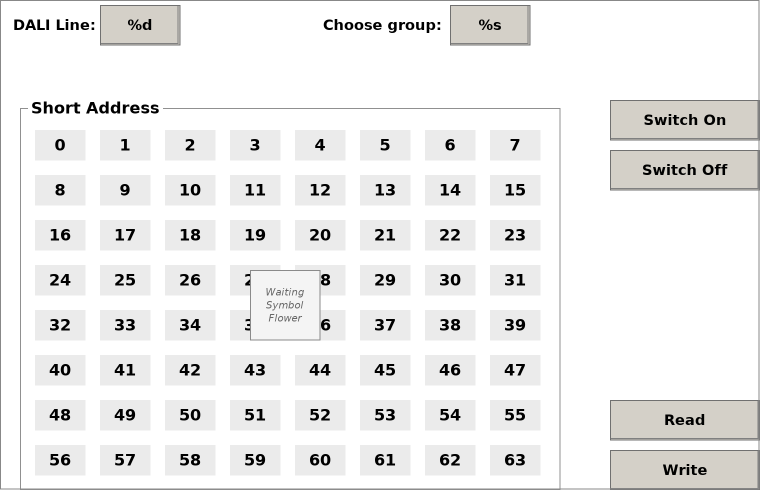
VISUALIZATION Visu_Part102Groups  // 760x490
    GroupBox (20,100 540x390), "Short Address"
        Textfield (15,30 50x30), "0", colour toggle: DALI_Commissioning.fbPart102Groups.aShowAlarmState[0] = TRUE, invisible if: DALI_Commissioning.fbPart102Groups.aActivateButton[0] = FALSE, input disabled if: DALI_Commissioning.fbPart102Groups.aActivateButton[0] = FALSE
            OnMouseClick: execute { DALI_Commissioning.fbPart102Groups.aButtonClick[0] := TRUE; }
        Textfield (80,30 50x30), "1", colour toggle: DALI_Commissioning.fbPart102Groups.aShowAlarmState[1] = TRUE, invisible if: DALI_Commissioning.fbPart102Groups.aActivateButton[1] = FALSE, input disabled if: DALI_Commissioning.fbPart102Groups.aActivateButton[1] = FALSE
            OnMouseClick: execute { DALI_Commissioning.fbPart102Groups.aButtonClick[1] := TRUE; }
        Textfield (145,30 50x30), "2", colour toggle: DALI_Commissioning.fbPart102Groups.aShowAlarmState[2] = TRUE, invisible if: DALI_Commissioning.fbPart102Groups.aActivateButton[2] = FALSE, input disabled if: DALI_Commissioning.fbPart102Groups.aActivateButton[2] = FALSE
            OnMouseClick: execute { DALI_Commissioning.fbPart102Groups.aButtonClick[2] := TRUE; }
        Textfield (210,30 50x30), "3", colour toggle: DALI_Commissioning.fbPart102Groups.aShowAlarmState[3] = TRUE, invisible if: DALI_Commissioning.fbPart102Groups.aActivateButton[3] = FALSE, input disabled if: DALI_Commissioning.fbPart102Groups.aActivateButton[3] = FALSE
            OnMouseClick: execute { DALI_Commissioning.fbPart102Groups.aButtonClick[3] := TRUE; }
        Textfield (275,30 50x30), "4", colour toggle: DALI_Commissioning.fbPart102Groups.aShowAlarmState[4] = TRUE, invisible if: DALI_Commissioning.fbPart102Groups.aActivateButton[4] = FALSE, input disabled if: DALI_Commissioning.fbPart102Groups.aActivateButton[4] = FALSE
            OnMouseClick: execute { DALI_Commissioning.fbPart102Groups.aButtonClick[4] := TRUE; }
        Textfield (340,30 50x30), "5", colour toggle: DALI_Commissioning.fbPart102Groups.aShowAlarmState[5] = TRUE, invisible if: DALI_Commissioning.fbPart102Groups.aActivateButton[5] = FALSE, input disabled if: DALI_Commissioning.fbPart102Groups.aActivateButton[5] = FALSE
            OnMouseClick: execute { DALI_Commissioning.fbPart102Groups.aButtonClick[5] := TRUE; }
        Textfield (405,30 50x30), "6", colour toggle: DALI_Commissioning.fbPart102Groups.aShowAlarmState[6] = TRUE, invisible if: DALI_Commissioning.fbPart102Groups.aActivateButton[6] = FALSE, input disabled if: DALI_Commissioning.fbPart102Groups.aActivateButton[6] = FALSE
            OnMouseClick: execute { DALI_Commissioning.fbPart102Groups.aButtonClick[6] := TRUE; }
        Textfield (470,30 50x30), "7", colour toggle: DALI_Commissioning.fbPart102Groups.aShowAlarmState[7] = TRUE, invisible if: DALI_Commissioning.fbPart102Groups.aActivateButton[7] = FALSE, input disabled if: DALI_Commissioning.fbPart102Groups.aActivateButton[7] = FALSE
            OnMouseClick: execute { DALI_Commissioning.fbPart102Groups.aButtonClick[7] := TRUE; }
        Textfield (15,75 50x30), "8", colour toggle: DALI_Commissioning.fbPart102Groups.aShowAlarmState[8] = TRUE, invisible if: DALI_Commissioning.fbPart102Groups.aActivateButton[8] = FALSE, input disabled if: DALI_Commissioning.fbPart102Groups.aActivateButton[8] = FALSE
            OnMouseClick: execute { DALI_Commissioning.fbPart102Groups.aButtonClick[8] := TRUE; }
        Textfield (80,75 50x30), "9", colour toggle: DALI_Commissioning.fbPart102Groups.aShowAlarmState[9] = TRUE, invisible if: DALI_Commissioning.fbPart102Groups.aActivateButton[9] = FALSE, input disabled if: DALI_Commissioning.fbPart102Groups.aActivateButton[9] = FALSE
            OnMouseClick: execute { DALI_Commissioning.fbPart102Groups.aButtonClick[9] := TRUE; }
        Textfield (145,75 50x30), "10", colour toggle: DALI_Commissioning.fbPart102Groups.aShowAlarmState[10] = TRUE, invisible if: DALI_Commissioning.fbPart102Groups.aActivateButton[10] = FALSE, input disabled if: DALI_Commissioning.fbPart102Groups.aActivateButton[10] = FALSE
            OnMouseClick: execute { DALI_Commissioning.fbPart102Groups.aButtonClick[10] := TRUE; }
        Textfield (210,75 50x30), "11", colour toggle: DALI_Commissioning.fbPart102Groups.aShowAlarmState[11] = TRUE, invisible if: DALI_Commissioning.fbPart102Groups.aActivateButton[11] = FALSE, input disabled if: DALI_Commissioning.fbPart102Groups.aActivateButton[11] = FALSE
            OnMouseClick: execute { DALI_Commissioning.fbPart102Groups.aButtonClick[11] := TRUE; }
        Textfield (275,75 50x30), "12", colour toggle: DALI_Commissioning.fbPart102Groups.aShowAlarmState[12] = TRUE, invisible if: DALI_Commissioning.fbPart102Groups.aActivateButton[12] = FALSE, input disabled if: DALI_Commissioning.fbPart102Groups.aActivateButton[12] = FALSE
            OnMouseClick: execute { DALI_Commissioning.fbPart102Groups.aButtonClick[12] := TRUE; }
        Textfield (340,75 50x30), "13", colour toggle: DALI_Commissioning.fbPart102Groups.aShowAlarmState[13] = TRUE, invisible if: DALI_Commissioning.fbPart102Groups.aActivateButton[13] = FALSE, input disabled if: DALI_Commissioning.fbPart102Groups.aActivateButton[13] = FALSE
            OnMouseClick: execute { DALI_Commissioning.fbPart102Groups.aButtonClick[13] := TRUE; }
        Textfield (405,75 50x30), "14", colour toggle: DALI_Commissioning.fbPart102Groups.aShowAlarmState[14] = TRUE, invisible if: DALI_Commissioning.fbPart102Groups.aActivateButton[14] = FALSE, input disabled if: DALI_Commissioning.fbPart102Groups.aActivateButton[14] = FALSE
            OnMouseClick: execute { DALI_Commissioning.fbPart102Groups.aButtonClick[14] := TRUE; }
        Textfield (470,75 50x30), "15", colour toggle: DALI_Commissioning.fbPart102Groups.aShowAlarmState[15] = TRUE, invisible if: DALI_Commissioning.fbPart102Groups.aActivateButton[15] = FALSE, input disabled if: DALI_Commissioning.fbPart102Groups.aActivateButton[15] = FALSE
            OnMouseClick: execute { DALI_Commissioning.fbPart102Groups.aButtonClick[15] := TRUE; }
        Textfield (15,120 50x30), "16", colour toggle: DALI_Commissioning.fbPart102Groups.aShowAlarmState[16] = TRUE, invisible if: DALI_Commissioning.fbPart102Groups.aActivateButton[16] = FALSE, input disabled if: DALI_Commissioning.fbPart102Groups.aActivateButton[16] = FALSE
            OnMouseClick: execute { DALI_Commissioning.fbPart102Groups.aButtonClick[16] := TRUE; }
        Textfield (80,120 50x30), "17", colour toggle: DALI_Commissioning.fbPart102Groups.aShowAlarmState[17] = TRUE, invisible if: DALI_Commissioning.fbPart102Groups.aActivateButton[17] = FALSE, input disabled if: DALI_Commissioning.fbPart102Groups.aActivateButton[17] = FALSE
            OnMouseClick: execute { DALI_Commissioning.fbPart102Groups.aButtonClick[17] := TRUE; }
        Textfield (145,120 50x30), "18", colour toggle: DALI_Commissioning.fbPart102Groups.aShowAlarmState[18] = TRUE, invisible if: DALI_Commissioning.fbPart102Groups.aActivateButton[18] = FALSE, input disabled if: DALI_Commissioning.fbPart102Groups.aActivateButton[18] = FALSE
            OnMouseClick: execute { DALI_Commissioning.fbPart102Groups.aButtonClick[18] := TRUE; }
        Textfield (210,120 50x30), "19", colour toggle: DALI_Commissioning.fbPart102Groups.aShowAlarmState[19] = TRUE, invisible if: DALI_Commissioning.fbPart102Groups.aActivateButton[19] = FALSE, input disabled if: DALI_Commissioning.fbPart102Groups.aActivateButton[19] = FALSE
            OnMouseClick: execute { DALI_Commissioning.fbPart102Groups.aButtonClick[19] := TRUE; }
        Textfield (275,120 50x30), "20", colour toggle: DALI_Commissioning.fbPart102Groups.aShowAlarmState[20] = TRUE, invisible if: DALI_Commissioning.fbPart102Groups.aActivateButton[20] = FALSE, input disabled if: DALI_Commissioning.fbPart102Groups.aActivateButton[20] = FALSE
            OnMouseClick: execute { DALI_Commissioning.fbPart102Groups.aButtonClick[20] := TRUE; }
        Textfield (340,120 50x30), "21", colour toggle: DALI_Commissioning.fbPart102Groups.aShowAlarmState[21] = TRUE, invisible if: DALI_Commissioning.fbPart102Groups.aActivateButton[21] = FALSE, input disabled if: DALI_Commissioning.fbPart102Groups.aActivateButton[21] = FALSE
            OnMouseClick: execute { DALI_Commissioning.fbPart102Groups.aButtonClick[21] := TRUE; }
        Textfield (405,120 50x30), "22", colour toggle: DALI_Commissioning.fbPart102Groups.aShowAlarmState[22] = TRUE, invisible if: DALI_Commissioning.fbPart102Groups.aActivateButton[22] = FALSE, input disabled if: DALI_Commissioning.fbPart102Groups.aActivateButton[22] = FALSE
            OnMouseClick: execute { DALI_Commissioning.fbPart102Groups.aButtonClick[22] := TRUE; }
        Textfield (470,120 50x30), "23", colour toggle: DALI_Commissioning.fbPart102Groups.aShowAlarmState[23] = TRUE, invisible if: DALI_Commissioning.fbPart102Groups.aActivateButton[23] = FALSE, input disabled if: DALI_Commissioning.fbPart102Groups.aActivateButton[23] = FALSE
            OnMouseClick: execute { DALI_Commissioning.fbPart102Groups.aButtonClick[23] := TRUE; }
        Textfield (15,165 50x30), "24", colour toggle: DALI_Commissioning.fbPart102Groups.aShowAlarmState[24] = TRUE, invisible if: DALI_Commissioning.fbPart102Groups.aDeviceGroupState[24] = 0, input disabled if: DALI_Commissioning.fbPart102Groups.aDeviceGroupState[24] = 0
            OnMouseClick: execute { DALI_Commissioning.fbPart102Groups.aButtonClick[24] := TRUE; }
        Textfield (80,165 50x30), "25", colour toggle: DALI_Commissioning.fbPart102Groups.aShowAlarmState[25] = TRUE, invisible if: DALI_Commissioning.fbPart102Groups.aActivateButton[25] = FALSE, input disabled if: DALI_Commissioning.fbPart102Groups.aActivateButton[25] = FALSE
            OnMouseClick: execute { DALI_Commissioning.fbPart102Groups.aButtonClick[25] := TRUE; }
        Textfield (145,165 50x30), "26", colour toggle: DALI_Commissioning.fbPart102Groups.aShowAlarmState[26] = TRUE, invisible if: DALI_Commissioning.fbPart102Groups.aActivateButton[26] = FALSE, input disabled if: DALI_Commissioning.fbPart102Groups.aActivateButton[26] = FALSE
            OnMouseClick: execute { DALI_Commissioning.fbPart102Groups.aButtonClick[26] := TRUE; }
        Textfield (210,165 50x30), "27", colour toggle: DALI_Commissioning.fbPart102Groups.aShowAlarmState[27] = TRUE, invisible if: DALI_Commissioning.fbPart102Groups.aActivateButton[27] = FALSE, input disabled if: DALI_Commissioning.fbPart102Groups.aActivateButton[27] = FALSE
            OnMouseClick: execute { DALI_Commissioning.fbPart102Groups.aButtonClick[27] := TRUE; }
        Textfield (275,165 50x30), "28", colour toggle: DALI_Commissioning.fbPart102Groups.aShowAlarmState[28] = TRUE, invisible if: DALI_Commissioning.fbPart102Groups.aActivateButton[28] = FALSE, input disabled if: DALI_Commissioning.fbPart102Groups.aActivateButton[28] = FALSE
            OnMouseClick: execute { DALI_Commissioning.fbPart102Groups.aButtonClick[28] := TRUE; }
        Textfield (340,165 50x30), "29", colour toggle: DALI_Commissioning.fbPart102Groups.aShowAlarmState[29] = TRUE, invisible if: DALI_Commissioning.fbPart102Groups.aActivateButton[29] = FALSE, input disabled if: DALI_Commissioning.fbPart102Groups.aActivateButton[29] = FALSE
            OnMouseClick: execute { DALI_Commissioning.fbPart102Groups.aButtonClick[29] := TRUE; }
        Textfield (405,165 50x30), "30", colour toggle: DALI_Commissioning.fbPart102Groups.aShowAlarmState[30] = TRUE, invisible if: DALI_Commissioning.fbPart102Groups.aActivateButton[30] = FALSE, input disabled if: DALI_Commissioning.fbPart102Groups.aActivateButton[30] = FALSE
            OnMouseClick: execute { DALI_Commissioning.fbPart102Groups.aButtonClick[30] := TRUE; }
        Textfield (470,165 50x30), "31", colour toggle: DALI_Commissioning.fbPart102Groups.aShowAlarmState[31] = TRUE, invisible if: DALI_Commissioning.fbPart102Groups.aActivateButton[31] = FALSE, input disabled if: DALI_Commissioning.fbPart102Groups.aActivateButton[31] = FALSE
            OnMouseClick: execute { DALI_Commissioning.fbPart102Groups.aButtonClick[31] := TRUE; }
        Textfield (15,210 50x30), "32", colour toggle: DALI_Commissioning.fbPart102Groups.aShowAlarmState[32] = TRUE, invisible if: DALI_Commissioning.fbPart102Groups.aActivateButton[32] = FALSE, input disabled if: DALI_Commissioning.fbPart102Groups.aActivateButton[32] = FALSE
            OnMouseClick: execute { DALI_Commissioning.fbPart102Groups.aButtonClick[32] := TRUE; }
        Textfield (80,210 50x30), "33", colour toggle: DALI_Commissioning.fbPart102Groups.aShowAlarmState[33] = TRUE, invisible if: DALI_Commissioning.fbPart102Groups.aActivateButton[33] = FALSE, input disabled if: DALI_Commissioning.fbPart102Groups.aActivateButton[33] = FALSE
            OnMouseClick: execute { DALI_Commissioning.fbPart102Groups.aButtonClick[33] := TRUE; }
        Textfield (145,210 50x30), "34", colour toggle: DALI_Commissioning.fbPart102Groups.aShowAlarmState[34] = TRUE, invisible if: DALI_Commissioning.fbPart102Groups.aActivateButton[34] = FALSE, input disabled if: DALI_Commissioning.fbPart102Groups.aActivateButton[34] = FALSE
            OnMouseClick: execute { DALI_Commissioning.fbPart102Groups.aButtonClick[34] := TRUE; }
        Textfield (210,210 50x30), "35", colour toggle: DALI_Commissioning.fbPart102Groups.aShowAlarmState[35] = TRUE, invisible if: DALI_Commissioning.fbPart102Groups.aActivateButton[35] = FALSE, input disabled if: DALI_Commissioning.fbPart102Groups.aActivateButton[35] = FALSE
            OnMouseClick: execute { DALI_Commissioning.fbPart102Groups.aButtonClick[35] := TRUE; }
        Textfield (275,210 50x30), "36", colour toggle: DALI_Commissioning.fbPart102Groups.aShowAlarmState[36] = TRUE, invisible if: DALI_Commissioning.fbPart102Groups.aActivateButton[36] = FALSE, input disabled if: DALI_Commissioning.fbPart102Groups.aActivateButton[36] = FALSE
            OnMouseClick: execute { DALI_Commissioning.fbPart102Groups.aButtonClick[36] := TRUE; }
        Textfield (340,210 50x30), "37", colour toggle: DALI_Commissioning.fbPart102Groups.aShowAlarmState[37] = TRUE, invisible if: DALI_Commissioning.fbPart102Groups.aActivateButton[37] = FALSE, input disabled if: DALI_Commissioning.fbPart102Groups.aActivateButton[37] = FALSE
            OnMouseClick: execute { DALI_Commissioning.fbPart102Groups.aButtonClick[37] := TRUE; }
        Textfield (405,210 50x30), "38", colour toggle: DALI_Commissioning.fbPart102Groups.aShowAlarmState[38] = TRUE, invisible if: DALI_Commissioning.fbPart102Groups.aActivateButton[38] = FALSE, input disabled if: DALI_Commissioning.fbPart102Groups.aActivateButton[38] = FALSE
            OnMouseClick: execute { DALI_Commissioning.fbPart102Groups.aButtonClick[38] := TRUE; }
        Textfield (470,210 50x30), "39", colour toggle: DALI_Commissioning.fbPart102Groups.aShowAlarmState[39] = TRUE, invisible if: DALI_Commissioning.fbPart102Groups.aActivateButton[39] = FALSE, input disabled if: DALI_Commissioning.fbPart102Groups.aActivateButton[39] = FALSE
            OnMouseClick: execute { DALI_Commissioning.fbPart102Groups.aButtonClick[39] := TRUE; }
        Textfield (15,255 50x30), "40", colour toggle: DALI_Commissioning.fbPart102Groups.aShowAlarmState[40] = TRUE, invisible if: DALI_Commissioning.fbPart102Groups.aActivateButton[40] = FALSE, input disabled if: DALI_Commissioning.fbPart102Groups.aActivateButton[40] = FALSE
            OnMouseClick: execute { DALI_Commissioning.fbPart102Groups.aButtonClick[40] := TRUE; }
        Textfield (80,255 50x30), "41", colour toggle: DALI_Commissioning.fbPart102Groups.aShowAlarmState[41] = TRUE, invisible if: DALI_Commissioning.fbPart102Groups.aActivateButton[41] = FALSE, input disabled if: DALI_Commissioning.fbPart102Groups.aActivateButton[41] = FALSE
            OnMouseClick: execute { DALI_Commissioning.fbPart102Groups.aButtonClick[41] := TRUE; }
        Textfield (145,255 50x30), "42", colour toggle: DALI_Commissioning.fbPart102Groups.aShowAlarmState[42] = TRUE, invisible if: DALI_Commissioning.fbPart102Groups.aActivateButton[42] = FALSE, input disabled if: DALI_Commissioning.fbPart102Groups.aActivateButton[42] = FALSE
            OnMouseClick: execute { DALI_Commissioning.fbPart102Groups.aButtonClick[42] := TRUE; }
        Textfield (210,255 50x30), "43", colour toggle: DALI_Commissioning.fbPart102Groups.aShowAlarmState[43] = TRUE, invisible if: DALI_Commissioning.fbPart102Groups.aActivateButton[43] = FALSE, input disabled if: DALI_Commissioning.fbPart102Groups.aActivateButton[43] = FALSE
            OnMouseClick: execute { DALI_Commissioning.fbPart102Groups.aButtonClick[43] := TRUE; }
        Textfield (275,255 50x30), "44", colour toggle: DALI_Commissioning.fbPart102Groups.aShowAlarmState[44] = TRUE, invisible if: DALI_Commissioning.fbPart102Groups.aActivateButton[44] = FALSE, input disabled if: DALI_Commissioning.fbPart102Groups.aActivateButton[44] = FALSE
            OnMouseClick: execute { DALI_Commissioning.fbPart102Groups.aButtonClick[44] := TRUE; }
        Textfield (340,255 50x30), "45", colour toggle: DALI_Commissioning.fbPart102Groups.aShowAlarmState[45] = TRUE, invisible if: DALI_Commissioning.fbPart102Groups.aActivateButton[45] = FALSE, input disabled if: DALI_Commissioning.fbPart102Groups.aActivateButton[45] = FALSE
            OnMouseClick: execute { DALI_Commissioning.fbPart102Groups.aButtonClick[45] := TRUE; }
        Textfield (405,255 50x30), "46", colour toggle: DALI_Commissioning.fbPart102Groups.aShowAlarmState[46] = TRUE, invisible if: DALI_Commissioning.fbPart102Groups.aActivateButton[46] = FALSE, input disabled if: DALI_Commissioning.fbPart102Groups.aActivateButton[46] = FALSE
            OnMouseClick: execute { DALI_Commissioning.fbPart102Groups.aButtonClick[46] := TRUE; }
        Textfield (470,255 50x30), "47", colour toggle: DALI_Commissioning.fbPart102Groups.aShowAlarmState[47] = TRUE, invisible if: DALI_Commissioning.fbPart102Groups.aActivateButton[47] = FALSE, input disabled if: DALI_Commissioning.fbPart102Groups.aActivateButton[47] = FALSE
            OnMouseClick: execute { DALI_Commissioning.fbPart102Groups.aButtonClick[47] := TRUE; }
        Textfield (15,300 50x30), "48", colour toggle: DALI_Commissioning.fbPart102Groups.aShowAlarmState[48] = TRUE, invisible if: DALI_Commissioning.fbPart102Groups.aActivateButton[48] = FALSE, input disabled if: DALI_Commissioning.fbPart102Groups.aActivateButton[48] = FALSE
            OnMouseClick: execute { DALI_Commissioning.fbPart102Groups.aButtonClick[48] := TRUE; }
        Textfield (80,300 50x30), "49", colour toggle: DALI_Commissioning.fbPart102Groups.aShowAlarmState[49] = TRUE, invisible if: DALI_Commissioning.fbPart102Groups.aActivateButton[49] = FALSE, input disabled if: DALI_Commissioning.fbPart102Groups.aActivateButton[49] = FALSE
            OnMouseClick: execute { DALI_Commissioning.fbPart102Groups.aButtonClick[49] := TRUE; }
        Textfield (145,300 50x30), "50", colour toggle: DALI_Commissioning.fbPart102Groups.aShowAlarmState[50] = TRUE, invisible if: DALI_Commissioning.fbPart102Groups.aActivateButton[50] = FALSE, input disabled if: DALI_Commissioning.fbPart102Groups.aActivateButton[50] = FALSE
            OnMouseClick: execute { DALI_Commissioning.fbPart102Groups.aButtonClick[50] := TRUE; }
        Textfield (210,300 50x30), "51", colour toggle: DALI_Commissioning.fbPart102Groups.aShowAlarmState[51] = TRUE, invisible if: DALI_Commissioning.fbPart102Groups.aActivateButton[51] = FALSE, input disabled if: DALI_Commissioning.fbPart102Groups.aActivateButton[51] = FALSE
            OnMouseClick: execute { DALI_Commissioning.fbPart102Groups.aButtonClick[51] := TRUE; }
        Textfield (275,300 50x30), "52", colour toggle: DALI_Commissioning.fbPart102Groups.aShowAlarmState[52] = TRUE, invisible if: DALI_Commissioning.fbPart102Groups.aActivateButton[52] = FALSE, input disabled if: DALI_Commissioning.fbPart102Groups.aActivateButton[52] = FALSE
            OnMouseClick: execute { DALI_Commissioning.fbPart102Groups.aButtonClick[52] := TRUE; }
        Textfield (340,300 50x30), "53", colour toggle: DALI_Commissioning.fbPart102Groups.aShowAlarmState[53] = TRUE, invisible if: DALI_Commissioning.fbPart102Groups.aActivateButton[53] = FALSE, input disabled if: DALI_Commissioning.fbPart102Groups.aActivateButton[53] = FALSE
            OnMouseClick: execute { DALI_Commissioning.fbPart102Groups.aButtonClick[53] := TRUE; }
        Textfield (405,300 50x30), "54", colour toggle: DALI_Commissioning.fbPart102Groups.aShowAlarmState[54] = TRUE, invisible if: DALI_Commissioning.fbPart102Groups.aActivateButton[54] = FALSE, input disabled if: DALI_Commissioning.fbPart102Groups.aActivateButton[54] = FALSE
            OnMouseClick: execute { DALI_Commissioning.fbPart102Groups.aButtonClick[54] := TRUE; }
        Textfield (470,300 50x30), "55", colour toggle: DALI_Commissioning.fbPart102Groups.aShowAlarmState[55] = TRUE, invisible if: DALI_Commissioning.fbPart102Groups.aActivateButton[55] = FALSE, input disabled if: DALI_Commissioning.fbPart102Groups.aActivateButton[55] = FALSE
            OnMouseClick: execute { DALI_Commissioning.fbPart102Groups.aButtonClick[55] := TRUE; }
        Textfield (15,345 50x30), "56", colour toggle: DALI_Commissioning.fbPart102Groups.aShowAlarmState[56] = TRUE, invisible if: DALI_Commissioning.fbPart102Groups.aActivateButton[56] = FALSE, input disabled if: DALI_Commissioning.fbPart102Groups.aActivateButton[56] = FALSE
            OnMouseClick: execute { DALI_Commissioning.fbPart102Groups.aButtonClick[56] := TRUE; }
        Textfield (80,345 50x30), "57", colour toggle: DALI_Commissioning.fbPart102Groups.aShowAlarmState[57] = TRUE, invisible if: DALI_Commissioning.fbPart102Groups.aActivateButton[57] = FALSE, input disabled if: DALI_Commissioning.fbPart102Groups.aActivateButton[57] = FALSE
            OnMouseClick: execute { DALI_Commissioning.fbPart102Groups.aButtonClick[56] := TRUE; }
        Textfield (145,345 50x30), "58", colour toggle: DALI_Commissioning.fbPart102Groups.aShowAlarmState[58] = TRUE, invisible if: DALI_Commissioning.fbPart102Groups.aActivateButton[58] = FALSE, input disabled if: DALI_Commissioning.fbPart102Groups.aActivateButton[58] = FALSE
            OnMouseClick: execute { DALI_Commissioning.fbPart102Groups.aButtonClick[58] := TRUE; }
        Textfield (210,345 50x30), "59", colour toggle: DALI_Commissioning.fbPart102Groups.aShowAlarmState[59] = TRUE, invisible if: DALI_Commissioning.fbPart102Groups.aActivateButton[59] = FALSE, input disabled if: DALI_Commissioning.fbPart102Groups.aActivateButton[59] = FALSE
            OnMouseClick: execute { DALI_Commissioning.fbPart102Groups.aButtonClick[59] := TRUE; }
        Textfield (275,345 50x30), "60", colour toggle: DALI_Commissioning.fbPart102Groups.aShowAlarmState[60] = TRUE, invisible if: DALI_Commissioning.fbPart102Groups.aActivateButton[60] = FALSE, input disabled if: DALI_Commissioning.fbPart102Groups.aActivateButton[60] = FALSE
            OnMouseClick: execute { DALI_Commissioning.fbPart102Groups.aButtonClick[60] := TRUE; }
        Textfield (340,345 50x30), "61", colour toggle: DALI_Commissioning.fbPart102Groups.aShowAlarmState[61] = TRUE, invisible if: DALI_Commissioning.fbPart102Groups.aActivateButton[61] = FALSE, input disabled if: DALI_Commissioning.fbPart102Groups.aActivateButton[61] = FALSE
            OnMouseClick: execute { DALI_Commissioning.fbPart102Groups.aButtonClick[61] := TRUE; }
        Textfield (405,345 50x30), "62", colour toggle: DALI_Commissioning.fbPart102Groups.aShowAlarmState[62] = TRUE, invisible if: DALI_Commissioning.fbPart102Groups.aActivateButton[62] = FALSE, input disabled if: DALI_Commissioning.fbPart102Groups.aActivateButton[62] = FALSE
            OnMouseClick: execute { DALI_Commissioning.fbPart102Groups.aButtonClick[62] := TRUE; }
        Textfield (470,345 50x30), "63", colour toggle: DALI_Commissioning.fbPart102Groups.aShowAlarmState[63] = TRUE, invisible if: DALI_Commissioning.fbPart102Groups.aActivateButton[63] = FALSE, input disabled if: DALI_Commissioning.fbPart102Groups.aActivateButton[63] = FALSE
            OnMouseClick: execute { DALI_Commissioning.fbPart102Groups.aButtonClick[63] := TRUE; }
        WaitingSymbolFlower (230,170 70x70), invisible if: DALI_Commissioning.fbPart102Groups.bHideWaitSymbol
    Button (610,400 150x40), "Read"
        OnMouseClick: execute { DALI_Commissioning.fbPart102Groups.bRead := TRUE; }
    Button (610,450 150x40), "Write"
        OnMouseClick: execute { DALI_Commissioning.fbPart102Groups.bWrite := TRUE; }
    Button (610,100 150x40), "Switch On"
        OnMouseClick: execute { DALI_Commissioning.fbPart102Groups.bSwitchOn := TRUE; }
    Button (610,150 150x40), "Switch Off"
        OnMouseClick: execute { DALI_Commissioning.fbPart102Groups.bSwitchOff := TRUE; }
    Group (320,5 210x40)
        Textfield (0,0 120x40), "Choose group:"
        Button (130,0 80x40), "%s", text variable: DALI_Commissioning.fbPart102Groups.nGroupAddress
            OnMouseClick: write the text variable via Default, min 0, max 15, title "Choose group"
    Group (10,5 170x40)
        Textfield (0,0 110x40), "DALI Line:"
        Button (90,0 80x40), "%d", text variable: GVL_Internal.nDALILine
            OnMouseClick: write the text variable via Default, min 1, max 10, title "Choose line"
END_VISUALIZATION

(* stored: Version 1.1.0.1
   Visu Visu_Part102Groups: Id {9fdf938c-2ad5-47f3-80cb-bc4b32517aaa} *)
